TYPE ST_6FDimm :
STRUCT
	sLocation			:STRING(28);	
	iDimm	 : ARRAY[1..6] OF INT;
END_STRUCT
END_TYPE

(* stored: Version 1.1.0.1, ProductVersion 3.1.4024.12
   DUT ST_6FDimm: Id {7a4b4ac1-55ba-4f20-b081-e433252ef29e} *)
